{attribute 'linkalways'} 
{attribute 'no_explicit_call' := 'This FB is a CLASS and must be accessed using methods or properties'}
{attribute 'enable_dynamic_creation'}
FUNCTION_BLOCK _ETcVnInitializableFunction EXTENDS EnumDatatypeBase
VAR
	localData : ETcVnInitializableFunction;
	activeData : REFERENCE TO ETcVnInitializableFunction;
	enumBaseDatatype : _DINT(localData);
END_VAR

METHOD PRIVATE AddLocalEnumeration
VAR_INPUT
	Enumeration : T_MAXSTRING;
	Value : ETcVnInitializableFunction;
END_VAR
AddEnumeration(Enumeration, Value);
END_METHOD

PROPERTY PUBLIC Address : PVOID
GET
Address := ADR(activeData);
END_GET
END_PROPERTY

METHOD PUBLIC ClearReference
VAR_INPUT
END_VAR
activeData REF= localData;
SetBaseDatatypeReference();
END_METHOD

METHOD PUBLIC Clone : I_Datatype
VAR
    pClone : POINTER TO _ETcVnInitializableFunction;
END_VAR
pClone := __NEW(_ETcVnInitializableFunction(InitialValue := Value));
Clone := pClone^;
END_METHOD

METHOD FB_init : BOOL
VAR_INPUT
	bInitRetains : BOOL; // if TRUE, the retain variables are initialized (warm start / cold start)
	bInCopyCode : BOOL;  // if TRUE, the instance afterwards gets moved into the copy code (online change)
	InitialValue : ETcVnInitializableFunction;
END_VAR
localData := InitialValue;
AddBaseDatatype(enumBaseDatatype);
ClearReference();

AddLocalEnumeration('TCVN_IF_OCR', ETcVnInitializableFunction.TCVN_IF_OCR);
END_METHOD

PROPERTY PUBLIC Identifier : T_MAXSTRING
GET
Identifier := 'ETcVnInitializableFunction';
END_GET
END_PROPERTY

METHOD IsEnumeratorValueEqual : BOOL
VAR_INPUT
	Enumerator : I_KeyValueForwardEnumerator;
END_VAR
VAR
	storedValue : ETcVnInitializableFunction;
END_VAR
IF NOT Enumerator.TryGet(storedValue) THEN
	RETURN;
END_IF

IsEnumeratorValueEqual := storedValue = activeData;
END_METHOD

METHOD PUBLIC MakeReferenceTo
VAR_INPUT
	ReferenceTarget : REFERENCE TO ETcVnInitializableFunction;
END_VAR
activeData REF= ReferenceTarget;
SetBaseDatatypeReference();
END_METHOD

METHOD PROTECTED SetBaseDatatypeReference
VAR_INPUT
END_VAR
enumBaseDatatype.MakeReferenceTo(activeData);
END_METHOD

PROPERTY PUBLIC Size : UDINT
GET
Size := SIZEOF(activeData);
END_GET
END_PROPERTY

METHOD TryMakeReferenceTo : BOOL
VAR_INPUT
	Target : I_Datatype;
END_VAR
VAR
	targetAsEnum : I_EnumDatatype;
	pTargetData : POINTER TO ETcVnInitializableFunction;
END_VAR
IF NOT Target.TryResolveAsEnumDatatype(targetAsEnum) THEN
	RETURN;
END_IF

IF targetAsEnum.Identifier <> Identifier THEN
	RETURN;
END_IF

pTargetData := Target.Address;
activeData REF= pTargetData^;
SetBaseDatatypeReference();
TryMakeReferenceTo := TRUE;
END_METHOD

PROPERTY PUBLIC Value : ETcVnInitializableFunction
GET
Value := activeData;
END_GET
SET
activeData := Value;
END_SET
END_PROPERTY

END_FUNCTION_BLOCK

(* stored: Version 1.1.0.1
   POU _ETcVnInitializableFunction: Id {a726ea83-3b67-4ca7-97e6-5c2a25c54afd}, SpecialFunc None
   Folder Constructor: Id {43d7c3f4-8d34-4772-9e1b-fe85e8820804}
   Folder Private: Id {fe4c3f96-901d-43c7-b3e1-158571905bfe}
   Folder Protected: Id {1ad56614-17df-45ba-8361-02380bc0affd}
   Method AddLocalEnumeration: Id {25adc8ba-4208-4e28-a4b2-9dd2142b6837}
   Property Address: Id {3f9835de-f453-455b-8d4a-55cc767a4dcf}
   Get Get: Id {53129a09-92d6-46e8-b1eb-0dcf4d977562}
   Method ClearReference: Id {0bc8d746-5106-4eb3-ac80-408fe33aaf13}
   Method Clone: Id {43d648a8-98d5-4b3f-bab2-11c1f4d6b61d}
   Method FB_init: Id {adf28df4-60d2-4e2c-ad2a-510f68a47dcc}
   Property Identifier: Id {baeb2000-cde2-43f5-86b9-31efc26538f0}
   Get Get: Id {f3fee34b-9c68-4103-81cc-9b5e20fdb565}
   Method IsEnumeratorValueEqual: Id {5ef327d7-9d07-42ce-9802-a84fcbeaa6ad}
   Method MakeReferenceTo: Id {863a98d5-b509-4fc6-aa90-e8f7a148d033}
   Method SetBaseDatatypeReference: Id {b94294b5-51ba-4af0-9136-3059e6da6367}
   Property Size: Id {5c51784f-74ad-4052-9bb9-e84b71756462}
   Get Get: Id {3fb9f855-648d-4940-9b54-35a262d4eaed}
   Method TryMakeReferenceTo: Id {14125601-7a08-4f1c-a36b-833e3af308f3}
   Property Value: Id {7a43dd33-d3a0-4ff0-944b-5d44d20f539e}
   Get Get: Id {62dd4970-4001-425b-8f50-2d4c385f57de}
   Set Set: Id {214bee76-173a-462b-b8f4-e305870dcc68} *)
